// ---- DUTs/IO/Topology/Beckhoff_EJ7xxxEK1122_3A43B222.TcDUT
{attribute 'GeneratedUsingTerminal: EK1122-0000-0018'}
{attribute addProperty BoxType "EK1122-0000-0018"}
{attribute addProperty Id "Beckhoff_EJ7xxxsub_EK1100EK1100_1FC0878B2"}
{attribute addProperty CRC "977515042"}
{attribute addProperty Size "2"}
{attribute addProperty Name "Beckhoff EJ7xxxEK1122"}
TYPE Beckhoff_EJ7xxxEK1122_3A43B222 EXTENDS EK1122_1FC0878B :
STRUCT
	{attribute addProperty Name "Beckhoff EJ7xxxsub EK1100"}
	{attribute addProperty PreviousPort "Beckhoff EJ7xxxEK1122 : D"}
	Beckhoff_EJ7xxxsub_EK1100 : EK1100_1FC0878B;
END_STRUCT
END_TYPE

// ---- DUTs/IO/Topology/Beckhoff_EJ7xxx_D0F87F47.TcDUT
{attribute 'GeneratedUsingTerminal: EK1100-0000-0018'}
{attribute addProperty BoxType "EK1100-0000-0018"}
{attribute addProperty Id "Beckhoff_EJ7xxxEK1122Beckhoff_EJ7xxxEK1122_3A43B2222A_0001_EJ7031_0000_0026EJ7031_022B480446A_0002_EJ7037_0000_0020EJ7037_3E4BEAEF54A_0003_EJ7041_0052_0016EJ7041_022B480446A_0004_EJ7047_0000_0018EJ7047_3E4BEAEF54A_0005_EJ7047_0000_0019EJ7047_3E4BEAEF54A_0006_EJ7047_0000_0020EJ7047_3E4BEAEF54A_0007_EJ7342_0000_0019EJ7342_2AE9C6B386A_0008_EJ7342_0000_0020EJ7342_2AE9C6B386A_0009_EJ7211_0010_0026EJ7211_CE650BCF33A_0010_EJ7211_0010_0027EJ7211_CE650BCF33A_0011_EJ7211_0010_0028EJ7211_CE650BCF33A_0012_EJ7211_0010_0029EJ7211_CE650BCF33A_0013_EJ7211_0010_0030EJ7211_FC4732E834A_0014_EJ7211_0010_0031EJ7211_FC4732E834A_0015_EJ7211_0010_0032EJ7211_FC4732E834A_0016_EJ7211_0011_0026EJ7211_7BF2131733A_0017_EJ7211_0011_0027EJ7211_7BF2131733A_0018_EJ7211_0011_0028EJ7211_7BF2131733A_0019_EJ7211_0011_0029EJ7211_7BF2131733A_0020_EJ7211_0011_0030EJ7211_7BF2131733A_0021_EJ7211_0011_0031EJ7211_7BF2131733A_0022_EJ7211_0011_0032EJ7211_7BF2131733A_0023_EJ7211_9414_0029EJ7211_CE650BCF33A_0024_EJ7211_9414_0030EJ7211_B7F6AF5335A_0025_EJ7211_9414_0031EJ7211_B7F6AF5335A_0026_EJ7211_9414_0032EJ7211_B7F6AF5335A_0027_EJ7211_9415_0029EJ7211_7BF2131733A_0028_EJ7211_9415_0030EJ7211_7BF2131733A_0029_EJ7211_9415_0031EJ7211_7BF2131733A_0030_EJ7211_9415_0032EJ7211_7BF2131733A_0031_EJ7334_0008_0016EJ7334_80FE8C1360A_0032_EJ7411_0000_0018EJ7411_236AD61B38"}
{attribute addProperty CRC "3505946439"}
{attribute addProperty Size "1315"}
{attribute addProperty Name "Beckhoff EJ7xxx"}
TYPE Beckhoff_EJ7xxx_D0F87F47 EXTENDS EK1100_1FC0878B :
STRUCT
	{attribute addProperty Name "Beckhoff EJ7xxxEK1122"}
	{attribute addProperty PreviousPort "Beckhoff EJ7xxx : B"}
	Beckhoff_EJ7xxxEK1122 : Beckhoff_EJ7xxxEK1122_3A43B222;
	{attribute addProperty Name "A_0001(EJ7031-0000-0026)"}
	{attribute addProperty PreviousPort "Beckhoff EJ7xxxEK1122 : C"}
	A_0001_EJ7031_0000_0026 : EJ7031_022B4804;
	{attribute addProperty Name "A_0002(EJ7037-0000-0020)"}
	{attribute addProperty PreviousPort "A_0001(EJ7031-0000-0026) : B"}
	A_0002_EJ7037_0000_0020 : EJ7037_3E4BEAEF;
	{attribute addProperty Name "A_0003(EJ7041-0052-0016)"}
	{attribute addProperty PreviousPort "A_0002(EJ7037-0000-0020) : B"}
	A_0003_EJ7041_0052_0016 : EJ7041_022B4804;
	{attribute addProperty Name "A_0004(EJ7047-0000-0018)"}
	{attribute addProperty PreviousPort "A_0003(EJ7041-0052-0016) : B"}
	A_0004_EJ7047_0000_0018 : EJ7047_3E4BEAEF;
	{attribute addProperty Name "A_0005(EJ7047-0000-0019)"}
	{attribute addProperty PreviousPort "A_0004(EJ7047-0000-0018) : B"}
	A_0005_EJ7047_0000_0019 : EJ7047_3E4BEAEF;
	{attribute addProperty Name "A_0006(EJ7047-0000-0020)"}
	{attribute addProperty PreviousPort "A_0005(EJ7047-0000-0019) : B"}
	A_0006_EJ7047_0000_0020 : EJ7047_3E4BEAEF;
	{attribute addProperty Name "A_0007(EJ7342-0000-0019)"}
	{attribute addProperty PreviousPort "A_0006(EJ7047-0000-0020) : B"}
	A_0007_EJ7342_0000_0019 : EJ7342_2AE9C6B3;
	{attribute addProperty Name "A_0008(EJ7342-0000-0020)"}
	{attribute addProperty PreviousPort "A_0007(EJ7342-0000-0019) : B"}
	A_0008_EJ7342_0000_0020 : EJ7342_2AE9C6B3;
	{attribute addProperty Name "A_0009(EJ7211-0010-0026)"}
	{attribute addProperty PreviousPort "A_0008(EJ7342-0000-0020) : B"}
	A_0009_EJ7211_0010_0026 : EJ7211_CE650BCF;
	{attribute addProperty Name "A_0010(EJ7211-0010-0027)"}
	{attribute addProperty PreviousPort "A_0009(EJ7211-0010-0026) : B"}
	A_0010_EJ7211_0010_0027 : EJ7211_CE650BCF;
	{attribute addProperty Name "A_0011(EJ7211-0010-0028)"}
	{attribute addProperty PreviousPort "A_0010(EJ7211-0010-0027) : B"}
	A_0011_EJ7211_0010_0028 : EJ7211_CE650BCF;
	{attribute addProperty Name "A_0012(EJ7211-0010-0029)"}
	{attribute addProperty PreviousPort "A_0011(EJ7211-0010-0028) : B"}
	A_0012_EJ7211_0010_0029 : EJ7211_CE650BCF;
	{attribute addProperty Name "A_0013(EJ7211-0010-0030)"}
	{attribute addProperty PreviousPort "A_0012(EJ7211-0010-0029) : B"}
	A_0013_EJ7211_0010_0030 : EJ7211_FC4732E8;
	{attribute addProperty Name "A_0014(EJ7211-0010-0031)"}
	{attribute addProperty PreviousPort "A_0013(EJ7211-0010-0030) : B"}
	A_0014_EJ7211_0010_0031 : EJ7211_FC4732E8;
	{attribute addProperty Name "A_0015(EJ7211-0010-0032)"}
	{attribute addProperty PreviousPort "A_0014(EJ7211-0010-0031) : B"}
	A_0015_EJ7211_0010_0032 : EJ7211_FC4732E8;
	{attribute addProperty Name "A_0016(EJ7211-0011-0026)"}
	{attribute addProperty PreviousPort "A_0015(EJ7211-0010-0032) : B"}
	A_0016_EJ7211_0011_0026 : EJ7211_7BF21317;
	{attribute addProperty Name "A_0017(EJ7211-0011-0027)"}
	{attribute addProperty PreviousPort "A_0016(EJ7211-0011-0026) : B"}
	A_0017_EJ7211_0011_0027 : EJ7211_7BF21317;
	{attribute addProperty Name "A_0018(EJ7211-0011-0028)"}
	{attribute addProperty PreviousPort "A_0017(EJ7211-0011-0027) : B"}
	A_0018_EJ7211_0011_0028 : EJ7211_7BF21317;
	{attribute addProperty Name "A_0019(EJ7211-0011-0029)"}
	{attribute addProperty PreviousPort "A_0018(EJ7211-0011-0028) : B"}
	A_0019_EJ7211_0011_0029 : EJ7211_7BF21317;
	{attribute addProperty Name "A_0020(EJ7211-0011-0030)"}
	{attribute addProperty PreviousPort "A_0019(EJ7211-0011-0029) : B"}
	A_0020_EJ7211_0011_0030 : EJ7211_7BF21317;
	{attribute addProperty Name "A_0021(EJ7211-0011-0031)"}
	{attribute addProperty PreviousPort "A_0020(EJ7211-0011-0030) : B"}
	A_0021_EJ7211_0011_0031 : EJ7211_7BF21317;
	{attribute addProperty Name "A_0022(EJ7211-0011-0032)"}
	{attribute addProperty PreviousPort "A_0021(EJ7211-0011-0031) : B"}
	A_0022_EJ7211_0011_0032 : EJ7211_7BF21317;
	{attribute addProperty Name "A_0023(EJ7211-9414-0029)"}
	{attribute addProperty PreviousPort "A_0022(EJ7211-0011-0032) : B"}
	A_0023_EJ7211_9414_0029 : EJ7211_CE650BCF;
	{attribute addProperty Name "A_0024(EJ7211-9414-0030)"}
	{attribute addProperty PreviousPort "A_0023(EJ7211-9414-0029) : B"}
	A_0024_EJ7211_9414_0030 : EJ7211_B7F6AF53;
	{attribute addProperty Name "A_0025(EJ7211-9414-0031)"}
	{attribute addProperty PreviousPort "A_0024(EJ7211-9414-0030) : B"}
	A_0025_EJ7211_9414_0031 : EJ7211_B7F6AF53;
	{attribute addProperty Name "A_0026(EJ7211-9414-0032)"}
	{attribute addProperty PreviousPort "A_0025(EJ7211-9414-0031) : B"}
	A_0026_EJ7211_9414_0032 : EJ7211_B7F6AF53;
	{attribute addProperty Name "A_0027(EJ7211-9415-0029)"}
	{attribute addProperty PreviousPort "A_0026(EJ7211-9414-0032) : B"}
	A_0027_EJ7211_9415_0029 : EJ7211_7BF21317;
	{attribute addProperty Name "A_0028(EJ7211-9415-0030)"}
	{attribute addProperty PreviousPort "A_0027(EJ7211-9415-0029) : B"}
	A_0028_EJ7211_9415_0030 : EJ7211_7BF21317;
	{attribute addProperty Name "A_0029(EJ7211-9415-0031)"}
	{attribute addProperty PreviousPort "A_0028(EJ7211-9415-0030) : B"}
	A_0029_EJ7211_9415_0031 : EJ7211_7BF21317;
	{attribute addProperty Name "A_0030(EJ7211-9415-0032)"}
	{attribute addProperty PreviousPort "A_0029(EJ7211-9415-0031) : B"}
	A_0030_EJ7211_9415_0032 : EJ7211_7BF21317;
	{attribute addProperty Name "A_0031(EJ7334-0008-0016)"}
	{attribute addProperty PreviousPort "A_0030(EJ7211-9415-0032) : B"}
	A_0031_EJ7334_0008_0016 : EJ7334_80FE8C13;
	{attribute addProperty Name "A_0032(EJ7411-0000-0018)"}
	{attribute addProperty PreviousPort "A_0031(EJ7334-0008-0016) : B"}
	A_0032_EJ7411_0000_0018 : EJ7411_236AD61B;
END_STRUCT
END_TYPE

// ---- DUTs/IO/Topology/Beckhoff_EJ9xxxEK1122_C80E1DB3.TcDUT
{attribute 'GeneratedUsingTerminal: EK1122-0000-0018'}
{attribute addProperty BoxType "EK1122-0000-0018"}
{attribute addProperty Id "Beckhoff_EJ9xxxsub_EK1100EK1100_1FC0878B2"}
{attribute addProperty CRC "3356368307"}
{attribute addProperty Size "2"}
{attribute addProperty Name "Beckhoff EJ9xxxEK1122"}
TYPE Beckhoff_EJ9xxxEK1122_C80E1DB3 EXTENDS EK1122_1FC0878B :
STRUCT
	{attribute addProperty Name "Beckhoff EJ9xxxsub EK1100"}
	{attribute addProperty PreviousPort "Beckhoff EJ9xxxEK1122 : D"}
	Beckhoff_EJ9xxxsub_EK1100 : EK1100_1FC0878B;
END_STRUCT
END_TYPE

// ---- DUTs/IO/Topology/Beckhoff_EJ9xxx_428E1E12.TcDUT
{attribute 'GeneratedUsingTerminal: EK1100-0000-0018'}
{attribute addProperty BoxType "EK1100-0000-0018"}
{attribute addProperty Id "Beckhoff_EJ9xxxEK1122Beckhoff_EJ9xxxEK1122_C80E1DB32A_0001_EJ9001_0000_0016EJ9001_1FC0878B2A_0002_EJ9505_0000_0016EJ9505_19A4723D6A_0003_EJ9576_0000_0018EJ9576_6D7359CA28A_0004_EJ9576_0000_0019EJ9576_85AB580429A_0005_EJ9576_0000_0020EJ9576_1017F4A528A_0006_EJ9576_0000_0022EJ9576_C42142C629A_0007_EJ9400_0000EJ9400_B5091FDC0A_0008_EJ9404_0000EJ9404_A60D69000"}
{attribute addProperty CRC "1116610066"}
{attribute addProperty Size "124"}
{attribute addProperty Name "Beckhoff EJ9xxx"}
TYPE Beckhoff_EJ9xxx_428E1E12 EXTENDS EK1100_1FC0878B :
STRUCT
	{attribute addProperty Name "Beckhoff EJ9xxxEK1122"}
	{attribute addProperty PreviousPort "Beckhoff EJ9xxx : B"}
	Beckhoff_EJ9xxxEK1122 : Beckhoff_EJ9xxxEK1122_C80E1DB3;
	{attribute addProperty Name "A_0001(EJ9001-0000-0016)"}
	{attribute addProperty PreviousPort "Beckhoff EJ9xxxEK1122 : C"}
	A_0001_EJ9001_0000_0016 : EJ9001_1FC0878B;
	{attribute addProperty Name "A_0002(EJ9505-0000-0016)"}
	{attribute addProperty PreviousPort "A_0001(EJ9001-0000-0016) : B"}
	A_0002_EJ9505_0000_0016 : EJ9505_19A4723D;
	{attribute addProperty Name "A_0003(EJ9576-0000-0018)"}
	{attribute addProperty PreviousPort "A_0002(EJ9505-0000-0016) : B"}
	A_0003_EJ9576_0000_0018 : EJ9576_6D7359CA;
	{attribute addProperty Name "A_0004(EJ9576-0000-0019)"}
	{attribute addProperty PreviousPort "A_0003(EJ9576-0000-0018) : B"}
	A_0004_EJ9576_0000_0019 : EJ9576_85AB5804;
	{attribute addProperty Name "A_0005(EJ9576-0000-0020)"}
	{attribute addProperty PreviousPort "A_0004(EJ9576-0000-0019) : B"}
	A_0005_EJ9576_0000_0020 : EJ9576_1017F4A5;
	{attribute addProperty Name "A_0006(EJ9576-0000-0022)"}
	{attribute addProperty PreviousPort "A_0005(EJ9576-0000-0020) : B"}
	A_0006_EJ9576_0000_0022 : EJ9576_C42142C6;
	{attribute addProperty Name "A_0007 (EJ9400-0000)"}
	{attribute addProperty PreviousPort "A_0006(EJ9576-0000-0022) : B"}
	A_0007_EJ9400_0000 : EJ9400_B5091FDC;
	{attribute addProperty Name "A_0008 (EJ9404-0000)"}
	{attribute addProperty PreviousPort "A_0006(EJ9576-0000-0022) : B"}
	A_0008_EJ9404_0000 : EJ9404_A60D6900;
END_STRUCT
END_TYPE

// ---- DUTs/IO/Topology/Beckhoff_EJx9xxEK1122_EEA9E9F5.TcDUT
{attribute 'GeneratedUsingTerminal: EK1122-0000-0018'}
{attribute addProperty BoxType "EK1122-0000-0018"}
{attribute addProperty Id "Beckhoff_EJx9xxsub_EK1100EK1100_1FC0878B2"}
{attribute addProperty CRC "4004112885"}
{attribute addProperty Size "2"}
{attribute addProperty Name "Beckhoff EJx9xxEK1122"}
TYPE Beckhoff_EJx9xxEK1122_EEA9E9F5 EXTENDS EK1122_1FC0878B :
STRUCT
	{attribute addProperty Name "Beckhoff EJx9xxsub EK1100"}
	{attribute addProperty PreviousPort "Beckhoff EJx9xxEK1122 : D"}
	Beckhoff_EJx9xxsub_EK1100 : EK1100_1FC0878B;
END_STRUCT
END_TYPE

// ---- DUTs/IO/Topology/Beckhoff_EJx9xx_66D9432D.TcDUT
{attribute 'GeneratedUsingTerminal: EK1100-0000-0018'}
{attribute addProperty BoxType "EK1100-0000-0018"}
{attribute addProperty Id "Beckhoff_EJx9xxEK1122Beckhoff_EJx9xxEK1122_EEA9E9F52A_0001_EJ1914_0000_0017EJ1914_0821024F34A_0002_EJ1914_0000_0018EJ1914_0821024F34A_0003_EJ1918_0000_0017EJ1918_57845E7942A_0004_EJ1918_0000_0018EJ1918_57845E7942A_0005_EJ1957_0000_0017EJ1957_9A95FC5954A_0006_EJ1957_0000_0018EJ1957_9A95FC5954A_0007_EJ2914_0000_0017EJ2914_475777A038A_0008_EJ2914_0000_0018EJ2914_475777A038A_0009_EJ2918_0000_0017EJ2918_B661C90A48A_0010_EJ2918_0000_0018EJ2918_B661C90A48A_0011_EJ6910_0000_0018EJ6910_CD4DE20014A_0012_EJ6910_0000_0020EJ6910_CD4DE20014"}
{attribute addProperty CRC "1725514541"}
{attribute addProperty Size "462"}
{attribute addProperty Name "Beckhoff EJx9xx"}
TYPE Beckhoff_EJx9xx_66D9432D EXTENDS EK1100_1FC0878B :
STRUCT
	{attribute addProperty Name "Beckhoff EJx9xxEK1122"}
	{attribute addProperty PreviousPort "Beckhoff EJx9xx : B"}
	Beckhoff_EJx9xxEK1122 : Beckhoff_EJx9xxEK1122_EEA9E9F5;
	{attribute addProperty Name "A_0001(EJ1914-0000-0017)"}
	{attribute addProperty PreviousPort "Beckhoff EJx9xxEK1122 : C"}
	A_0001_EJ1914_0000_0017 : EJ1914_0821024F;
	{attribute addProperty Name "A_0002(EJ1914-0000-0018)"}
	{attribute addProperty PreviousPort "A_0001(EJ1914-0000-0017) : B"}
	A_0002_EJ1914_0000_0018 : EJ1914_0821024F;
	{attribute addProperty Name "A_0003(EJ1918-0000-0017)"}
	{attribute addProperty PreviousPort "A_0002(EJ1914-0000-0018) : B"}
	A_0003_EJ1918_0000_0017 : EJ1918_57845E79;
	{attribute addProperty Name "A_0004(EJ1918-0000-0018)"}
	{attribute addProperty PreviousPort "A_0003(EJ1918-0000-0017) : B"}
	A_0004_EJ1918_0000_0018 : EJ1918_57845E79;
	{attribute addProperty Name "A_0005(EJ1957-0000-0017)"}
	{attribute addProperty PreviousPort "A_0004(EJ1918-0000-0018) : B"}
	A_0005_EJ1957_0000_0017 : EJ1957_9A95FC59;
	{attribute addProperty Name "A_0006(EJ1957-0000-0018)"}
	{attribute addProperty PreviousPort "A_0005(EJ1957-0000-0017) : B"}
	A_0006_EJ1957_0000_0018 : EJ1957_9A95FC59;
	{attribute addProperty Name "A_0007(EJ2914-0000-0017)"}
	{attribute addProperty PreviousPort "A_0006(EJ1957-0000-0018) : B"}
	A_0007_EJ2914_0000_0017 : EJ2914_475777A0;
	{attribute addProperty Name "A_0008(EJ2914-0000-0018)"}
	{attribute addProperty PreviousPort "A_0007(EJ2914-0000-0017) : B"}
	A_0008_EJ2914_0000_0018 : EJ2914_475777A0;
	{attribute addProperty Name "A_0009(EJ2918-0000-0017)"}
	{attribute addProperty PreviousPort "A_0008(EJ2914-0000-0018) : B"}
	A_0009_EJ2918_0000_0017 : EJ2918_B661C90A;
	{attribute addProperty Name "A_0010(EJ2918-0000-0018)"}
	{attribute addProperty PreviousPort "A_0009(EJ2918-0000-0017) : B"}
	A_0010_EJ2918_0000_0018 : EJ2918_B661C90A;
	{attribute addProperty Name "A_0011(EJ6910-0000-0018)"}
	{attribute addProperty PreviousPort "A_0010(EJ2918-0000-0018) : B"}
	A_0011_EJ6910_0000_0018 : EJ6910_CD4DE200;
	{attribute addProperty Name "A_0012(EJ6910-0000-0020)"}
	{attribute addProperty PreviousPort "A_0011(EJ6910-0000-0018) : B"}
	A_0012_EJ6910_0000_0020 : EJ6910_CD4DE200;
END_STRUCT
END_TYPE

// ---- DUTs/IO/Topology/EtherCAT_Master_EJxxxx_F8B494BA.TcDUT
{attribute 'GeneratedUsingTerminal: IODEVICETYPE_ETHERCATPROT'}
{attribute addProperty BoxType "IODEVICETYPE_ETHERCATPROT"}
{attribute addProperty Id "Beckhoff_EJ1xxxBeckhoff_EJ1xxx_8ABA4DFB121Beckhoff_EJ2xxxBeckhoff_EJ2xxx_F745D3BC254Beckhoff_EJ3xxxBeckhoff_EJ3xxx_05F253C11180Beckhoff_EJ4xxxBeckhoff_EJ4xxx_77B5C5A6177Beckhoff_EJ5xxxBeckhoff_EJ5xxx_E1A62FB7142Beckhoff_EJ6xxxBeckhoff_EJ6xxx_D380D5DE176Beckhoff_EJ7xxxBeckhoff_EJ7xxx_D0F87F471315Beckhoff_EJ9xxxBeckhoff_EJ9xxx_428E1E12124Beckhoff_EJx9xxBeckhoff_EJx9xx_66D9432D462SyncUnitsSyncUnits_99E584AF18InputsInputs_25A0042B160OutputsOutputs_2397A10E106InfoDataInfoData_E68C61CD28"}
{attribute addProperty CRC "4172584122"}
{attribute addProperty Size "4263"}
{attribute addProperty Name "EtherCAT Master EJxxxx"}
TYPE EtherCAT_Master_EJxxxx_F8B494BA EXTENDS EtcMasterBase_62654B43 :
STRUCT
	{attribute addProperty Name "Beckhoff EJ1xxx"}
	{attribute addProperty PreviousPort "EtherCAT Master EJxxxx : Master"}
	Beckhoff_EJ1xxx : Beckhoff_EJ1xxx_8ABA4DFB;
	{attribute addProperty Name "Beckhoff EJ2xxx"}
	{attribute addProperty PreviousPort "Beckhoff EJ1xxx : C"}
	Beckhoff_EJ2xxx : Beckhoff_EJ2xxx_F745D3BC;
	{attribute addProperty Name "Beckhoff EJ3xxx"}
	{attribute addProperty PreviousPort "Beckhoff EJ2xxx : C"}
	Beckhoff_EJ3xxx : Beckhoff_EJ3xxx_05F253C1;
	{attribute addProperty Name "Beckhoff EJ4xxx"}
	{attribute addProperty PreviousPort "Beckhoff EJ3xxx : C"}
	Beckhoff_EJ4xxx : Beckhoff_EJ4xxx_77B5C5A6;
	{attribute addProperty Name "Beckhoff EJ5xxx"}
	{attribute addProperty PreviousPort "Beckhoff EJ4xxx : C"}
	Beckhoff_EJ5xxx : Beckhoff_EJ5xxx_E1A62FB7;
	{attribute addProperty Name "Beckhoff EJ6xxx"}
	{attribute addProperty PreviousPort "Beckhoff EJ5xxx : C"}
	Beckhoff_EJ6xxx : Beckhoff_EJ6xxx_D380D5DE;
	{attribute addProperty Name "Beckhoff EJ7xxx"}
	{attribute addProperty PreviousPort "Beckhoff EJ6xxx : C"}
	Beckhoff_EJ7xxx : Beckhoff_EJ7xxx_D0F87F47;
	{attribute addProperty Name "Beckhoff EJ9xxx"}
	{attribute addProperty PreviousPort "Beckhoff EJ7xxx : C"}
	Beckhoff_EJ9xxx : Beckhoff_EJ9xxx_428E1E12;
	{attribute addProperty Name "Beckhoff EJx9xx"}
	{attribute addProperty PreviousPort "Beckhoff EJ9xxx : C"}
	Beckhoff_EJx9xx : Beckhoff_EJx9xx_66D9432D;
	{attribute addProperty Name "SyncUnits"}
	SyncUnits : SyncUnits_99E584AF;
	{attribute addProperty Name "Inputs"}
	Inputs : Inputs_25A0042B;
	{attribute addProperty Name "Outputs"}
	Outputs : Outputs_2397A10E;
	{attribute addProperty Name "InfoData"}
	InfoData : InfoData_E68C61CD;
END_STRUCT
END_TYPE

// ---- DUTs/IO/Base/EtcSlaveBase_82538BE2.TcDUT

TYPE EtcSlaveBase_82538BE2 :
STRUCT
END_STRUCT
END_TYPE

// ---- DUTs/IO/Base/EtcSlaveBase_82538BE2.TcDUT

TYPE EtcSlaveBase_82538BE2 :
STRUCT
END_STRUCT
END_TYPE

// ---- DUTs/IO/Base/EtcSlaveBase_82538BE2.TcDUT

TYPE EtcSlaveBase_82538BE2 :
STRUCT
END_STRUCT
END_TYPE

// ---- DUTs/IO/Base/EtcSlaveTerminalBase_947E5A46.TcDUT

{attribute clr[Container(Layout.Stack)]}
{attribute clr[Group(Layout.GroupBox)]}
{attribute addProperty PreviousPort "Unknown"}
TYPE EtcSlaveTerminalBase_947E5A46 EXTENDS EtcSlaveBase_82538BE2 :
STRUCT
END_STRUCT
END_TYPE

// ---- DUTs/IO/Base/EtcSlaveBoxBase_77A0E4A7.TcDUT

{attribute clr[Container(Layout.Stack)]}
{attribute clr[Group(Layout.GroupBox)]}
{attribute addProperty PreviousPort "Unknown"}
TYPE EtcSlaveBoxBase_77A0E4A7 EXTENDS EtcSlaveBase_82538BE2 :
STRUCT
END_STRUCT
END_TYPE

// ---- DUTs/IO/Base/EtcSlaveEndTerminalBase_866C7F0C.TcDUT

{attribute clr[Container(Layout.Stack)]}
{attribute clr[Group(Layout.GroupBox)]}
{attribute addProperty PreviousPort "Unknown"}
TYPE EtcSlaveEndTerminalBase_866C7F0C EXTENDS EtcSlaveBase_82538BE2 :
STRUCT
END_STRUCT
END_TYPE

// ---- DUTs/IO/Base/InputBase_8311D824.TcDUT

TYPE InputBase_8311D824 :
STRUCT
END_STRUCT
END_TYPE

// ---- DUTs/IO/Base/OutputBase_10CEE7DE.TcDUT

TYPE OutputBase_10CEE7DE :
STRUCT
END_STRUCT
END_TYPE

// ---- DUTs/IO/Base/EtcMasterBase_62654B43.TcDUT

TYPE EtcMasterBase_62654B43 :
STRUCT
END_STRUCT
END_TYPE

// ---- GVLs/GVL_iXlinker.TcGVL
{attribute 'qualified_only'}
VAR_GLOBAL
		EtherCAT_Master_EJxxxx : EtherCAT_Master_EJxxxx_F8B494BA;
END_VAR

// ---- POUs/MAIN.TcPOU
PROGRAM MAIN
VAR
END_VAR

END_PROGRAM
